VAR_GLOBAL
	//B940-009-R17-PCI-03
	{attribute 'pytmc' := ' pv: TXI:PIP:01 '}
	fb_ST1L1_PIP_01: FB_PIP_GAMMA;
	st_ST1L1_PIP_01: ST_PIP;
	
END_VAR

(* stored: Version 1.1.0.1, ProductVersion 3.1.4024.6
   GVL GVL_TXI_VAC_PUMPS: Id {90b18ceb-1c3e-4845-8d8c-a86724f4d309} *)
